(* CoDeSys 2.3.9.35 project: p1q2.pro *)
(* Author: Hemerson *)
(* Libraries: SysLibTargetVisu.lib 26.11.08 09:50:36, Standard.lib 26.11.08 09:46:20, Iecsfc.lib 26.11.08 09:46:14, DU35x.lib 7.7.11 15:59:53, SYSLIBCALLBACK.LIB 26.11.08 09:50:38 *)

(* PLC configuration (modules and I/O channels)
MToolIEC [Codesys] node 0, in %IB0 out %QB0
COM2 [COM2] node 1, in %IB0 out %QB0 {BaudRate = 115200; Paridade = No Parity; StopBits = 1 Stop Bit; Modem = Without RTS/CTS; Delay = 5}
  Disable [Desabilitado485] node 0, in %IB0 out %QB0
Digital Inputs 0 [Entradas0] node 0, in %IW0 out %QB0
  I00 AT %IX0.0 [BitInput] I0.0
  I01 AT %IX0.1 [BitInput] I0.1
  I02 AT %IX0.2 [BitInput] I0.2
  I03 AT %IX0.3 [BitInput] I0.3
  I04 AT %IX0.4 [BitInput] I0.4
  I05 AT %IX0.5 [BitInput] I0.5
  I06 AT %IX0.6 [BitInput] I0.6
  I07 AT %IX0.7 [BitInput] I0.7
  I08 AT %IX0.8 [BitInput] I0.8
Digital Inputs 1 [Entradas1] node 0, in %IW1 out %QB0
  I10 AT %IX1.0 [BitInput] I1.0
  I11 AT %IX1.1 [BitInput] I1.1
  I12 AT %IX1.2 [BitInput] I1.2
  I13 AT %IX1.3 [BitInput] I1.3
  I14 AT %IX1.4 [BitInput] I1.4
  I15 AT %IX1.5 [BitInput] I1.5
  I16 AT %IX1.6 [BitInput] I1.6
  I17 AT %IX1.7 [BitInput] I1.7
  I18 AT %IX1.8 [BitInput] I1.8
Digital Inputs 2 [Entradas2] node 0, in %IW2 out %QB0
  I20 AT %IX2.0 [BitInput] I2.0
  I21 AT %IX2.1 [BitInput] I2.1
AI0 AT %IW4 [WordInput] AI0 {TipoAnalogica = Canal Desabilitado; FiltroAnalogica = Filtro 0 - AI=2ms  / AV=90ms; FundoEscala = 0}
AI1 AT %IW5 [WordInput] AI1 {TipoAnalogica = Channel Disable; FiltroAnalogica = Filter 0 - AI=2ms  / AV=90ms; FundoEscala = 0}
AI2 AT %IW6 [WordInput] AI2 {TipoAnalogica = Channel Disable; FiltroAnalogica = Filter 0 - AI=2ms  / AV=90ms; FundoEscala = 0}
AI3 AT %IW7 [WordInput] AI3 {TipoAnalogica = Channel Disable; FiltroAnalogica = Filter 0 - AI=2ms  / AV=90ms; FundoEscala = 0}
Fast Inputs [EntradasRapidas] node 1, in %IB16 out %QB0
  Block 0 [Bloco0] node 0, in %IB16 out %QB0
    Disable [DesabilitadoBloco0] node 0, in %IB16 out %QB0
  Block 1 [Bloco1] node 1, in %IB16 out %QB0
    Disable [DesabilitadoBloco1] node 0, in %IB16 out %QB0
  Configurable Input Block 0 [EntradaConfiBloco0] node 2, in %IB16 out %QB0
    Counter 0 [EntradaConfContador0] node 0, in %IB16 out %QB0 {EntradaConfiguravelContador = Disable}
  Configurable Input Block 1 [EntradaConfiBloco1] node 3, in %IB16 out %QB0
    Counter 2 [EntradaConfContador2] node 0, in %IB16 out %QB0 {EntradaConfiguravelContador = Disable}
Outputs [Saidas] node 1, in %IB13 out %QB0
  Digital Outputs 0 [Saidas0] node 0, in %IW0 out %QW0
    Q00 AT %QX0.0 [BitOutput] Q0.0
    Q01 AT %QX0.1 [BitOutput] Q0.1
    Q02 AT %QX0.2 [BitOutput] Q0.2
    Q03 AT %QX0.3 [BitOutput] Q0.3
    Q04 AT %QX0.4 [BitOutput] Q0.4
    Q05 AT %QX0.5 [BitOutput] Q0.5
    Q06 AT %QX0.6 [BitOutput] Q0.6
    Q07 AT %QX0.7 [BitOutput] Q0.7
  Digital Outputs 1 [Saidas1] node 0, in %IW0 out %QW1
    Q10 AT %QX1.0 [BitOutput] Q1.0
    Q11 AT %QX1.1 [BitOutput] Q1.1
    Q12 AT %QX1.2 [BitOutput] Q1.2
    Q13 AT %QX1.3 [BitOutput] Q1.3
    Q14 AT %QX1.4 [BitOutput] Q1.4
    Q15 AT %QX1.5 [BitOutput] Q1.5
    Q16 AT %QX1.6 [BitOutput] Q1.6
    Q17 AT %QX1.7 [BitOutput] Q1.7
  Analog Outputs [SaidaAnalogica] node 0, in %IW0 out %QW3
    AO0 AT %QW3 [WordOutput] AO0 {TipoAnalogica = Channel Disable; FundoEscala = 0}
    AO1 AT %QW4 [WordOutput] AO1 {TipoAnalogica = Channel Disable; FundoEscala = 0}
  Fast Outputs [SaidasRapidas] node 1, in %IB0 out %QB10
    Fast Output 0 Disable [DesabilitadoF0] node 0, in %IB0 out %QB10
    Fast Output 1 Disable [DesabilitadoF1] node 1, in %IB0 out %QB10
  Counter Output [SaidasContador] node 2, in %IB0 out %QB10
    Block 0 Output Disable [DesabilitadoSaidaBloco0] node 0, in %IB0 out %QB10
    Block 1 Output Disable [DesabilitadoSaidaBloco1] node 1, in %IB0 out %QB10
External Events [Eventos] node 2, in %IB13 out %QB6
  Timer Event [TimerEvent] node 0, in %IB13 out %QB6 {Intervalo = 10}
*)

(* Global variable list: Variáveis globais *)
VAR_GLOBAL
	I0 AT %IX0.0: BOOL;
	I1 AT %IX0.1: BOOL;
	I2 AT %IX0.2: BOOL;
	I3 AT %IX0.3: BOOL;
	I4 AT %IX0.4: BOOL;
	I5 AT %IX0.5: BOOL;
	O1 AT %QX1.1: BOOL;
	O2 AT %QX1.2: BOOL;
END_VAR

(* POU PLC_PRG, LD *)
PROGRAM PLC_PRG
VAR_INPUT
	I0 AT %IX0.0: BOOL;
	I1 AT %IX0.1: BOOL;
	I2 AT %IX0.2: BOOL;
	I3 AT %IX0.3: BOOL;
	I4 AT %IX0.4: BOOL;
	I5 AT %IX0.5: BOOL;
END_VAR
VAR_OUTPUT
	O1 AT %QX1.1: BOOL;
	O2 AT %QX1.2: BOOL;
END_VAR
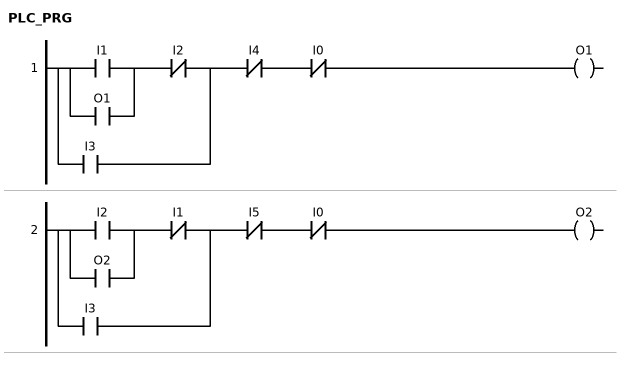
_LD_ (* Ladder Diagram *)
NETWORK 1
	{ { [I1] | [O1] } - [/I2] | [I3] } - [/I4] - [/I0] --- (O1)
NETWORK 2
	{ { [I2] | [O2] } - [/I1] | [I3] } - [/I5] - [/I0] --- (O2)
_END_LD_
(* the same logic as Structured Text *)
(* Network 1 *)
O1 := ((I1 OR O1) AND NOT I2 OR I3) AND NOT I4 AND NOT I0;
(* Network 2 *)
O2 := ((I2 OR O2) AND NOT I1 OR I3) AND NOT I5 AND NOT I0;
END_PROGRAM

(* Visualisation VP1Q1
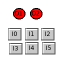
ellipse at (9,5)-(21,16): text "O1"; alarm colour if .O1
ellipse at (26,5)-(38,16): text "O2"; alarm colour if .O2
button at (4,25)-(17,37): text "I0"; toggles .I0
button at (21,25)-(34,37): text "I1"; toggles .I1
button at (37,25)-(50,37): text "I2"; toggles .I2
button at (5,40)-(18,51): text "I3"; toggles .I3
button at (21,39)-(34,51): text "I4"; toggles .I4
button at (38,39)-(51,51): text "I5"; toggles .I5
*)
